// TIA Portal V20 export
DATA_BLOCK "EmNodes"   // DB146
// Global DB for the data exchange between the module levels (Between Unit and EM or EM and CM)
// stored: Access Published, MemoryReserve 100, Namespace Unit1
   VAR
      unitStatus { ExternalWritable := 'False'} : "LAF_typeUnitStatus";   // Status of the unit
      emFeedback { ExternalWritable := 'False'} : Array[0.._.U1_NO_OF_EMs] of "LUC_typeEmFeedback";   // Status of the individual equipment modules
      emRelations { ExternalWritable := 'False'} : "Unit1.LER_typeEmRelation";
      emIt { S7_SetPoint := 'True'} : Array[0..13] of "LER_OEM_Data";
      enableControlInterfaces { ExternalWritable := 'False'} : "LAF_typeEnableControlInterfaces";
      oem { ExternalAccessible := 'False'; ExternalVisible := 'False'; ExternalWritable := 'False'; S7_SetPoint := 'True'} : Array[0..10] of "LER_OEM_Data";
      FATModeSelect { ExternalWritable := 'False'} : "LER_TypeFATMode_ModeSelect";
   END_VAR
   VAR RETAIN
      FATModeInterface { ExternalWritable := 'False'} : "LER_TypeFATModeInterface";
   END_VAR
   VAR
      signalStack { ExternalWritable := 'False'} : "LUC_typeSignalStackByBool";
      clock { ExternalWritable := 'False'} : "LAF_typeGlobalClockMem";
      slmRunning { ExternalWritable := 'False'} : Bool;
      slmPowerOff { ExternalWritable := 'False'} : Bool;
      InterfaceTestMode { ExternalWritable := 'False'} : Bool;
      CapabilityModeComplete { ExternalWritable := 'False'} : Bool;
      SamplingModeComplete { ExternalWritable := 'False'} : Bool;
      stateCommandsExecute { ExternalWritable := 'False'} : Bool;
      atLeastOneDoorUnLock { ExternalWritable := 'False'} : Bool;
      SleepModeActivationTime { ExternalWritable := 'False'} : Time;
      DeepSleepModeActivationTime { ExternalWritable := 'False'} : Time;
      SleepModeChangeReq { ExternalWritable := 'False'} : Bool;
      DeepSleepModeChangeReq { ExternalWritable := 'False'} : Bool;
      WakeupRecoveryRequired { ExternalWritable := 'False'} : Bool;
      "========Communication========" { ExternalWritable := 'False'} : Bool;
      BA030 { ExternalWritable := 'False'} : "LER_typeCommunication";
      BA040 { ExternalWritable := 'False'} : "LER_typeCommunication";
      "========Safety========" { ExternalWritable := 'False'} : Bool;
      devicesSummary { ExternalWritable := 'False'} : "LWONIK_typeDevicesStatusSummary";
      OperationMode { ExternalWritable := 'False'} : "LWONIK_typeOperationMode";
      PhmiMode { ExternalWritable := 'False'} : "LWONIK_typePhmiMode";
      ScsMode { ExternalWritable := 'False'} : "LWONIK_typeScsMode";
      RcMode1 { ExternalWritable := 'False'} : "LWONIK_typeRollChangeMode";
      RcMode2 { ExternalWritable := 'False'} : "LWONIK_typeRollChangeMode";
      SafetyZone1OpEnable { ExternalWritable := 'False'} : "LWONIK_typeSafetyZoneManualOperation";
      SafetyZone2OpEnable { ExternalWritable := 'False'} : "LWONIK_typeSafetyZoneManualOperation";
      SafetyZone3OpEnable { ExternalWritable := 'False'} : "LWONIK_typeSafetyZoneManualOperation";
      Zone1SafetyStatus { ExternalWritable := 'False'} : "LWONIK_typeZoneStatus";
      Zone2SafetyStatus { ExternalWritable := 'False'} : "LWONIK_typeZoneStatus";
      Zone3SafetyStatus { ExternalWritable := 'False'} : "LWONIK_typeZoneStatus";
      SafetySensor { ExternalWritable := 'False'} : "LWONIK_typeSafetySensor";
      EstopStatus { ExternalWritable := 'False'} : "LWONIK_typeFromSafetyEstopStatus";
      FdoorStatus { ExternalWritable := 'False'} : "LWONIK_typeFromSafetyDoorStatus";
      MobilePanelConnected { ExternalWritable := 'False'} : Bool;
      EnableACK { ExternalWritable := 'False'} : Bool;
      SS1Extention { ExternalWritable := 'False'} : Bool;
      LHSS1Extention { ExternalWritable := 'False'} : Bool;
      RHSS1Extention { ExternalWritable := 'False'} : Bool;
      LH_RollChangeActive { ExternalWritable := 'False'} : Bool;
      RH_RollChangeActive { ExternalWritable := 'False'} : Bool;
      Z_FOLD_AllEstopsOK { ExternalWritable := 'False'} : Bool;
      "=======ETC========" { ExternalWritable := 'False'} : Bool;
   END_VAR
   VAR RETAIN
      unitRecipe { ExternalWritable := 'False'} : "Unit1.typeRecipe";
   END_VAR
   VAR
      unitCycleTime { ExternalWritable := 'False'} : Time;
      "unitCycleTime/2" { ExternalWritable := 'False'} : Time;
      "unitCycleTime/6" { ExternalWritable := 'False'} : Time;
      allBrakeTest { ExternalWritable := 'False'} : "LER_typeBrakeTestUnitInterface";
      HourTestModeAllOK { ExternalWritable := 'False'} : Bool;
      CapabilityModeAllOK { ExternalWritable := 'False'} : Bool;
      ScrapBox { ExternalWritable := 'False'} : Struct
         LockSW : Bool;
         UnlockSW : Bool;
         ResetSW : Bool;
      END_STRUCT;
      LeftSafeScale { ExternalWritable := 'False'} : Int := 120;
      RightSafeScale { ExternalWritable := 'False'} : Int := 120;
      LeftMaxValue : Int := 1020;
      RightMaxValue : Int := 1020;
   END_VAR
BEGIN
   // BA030.ReelCutToStack.InterfaceData."Bool"[0] : To Load Enable
   // BA030.ReelCutToStack.InterfaceData."Bool"[1] : To Load Complete Comfirm
   // BA030.ReelCutToStack.InterfaceData."Bool"[2] : Cell Data Report
   // BA030.ReelCutToStack.InterfaceData."Bool"[10] : CollisionAreaOn
   // BA030.ReelCutToStack.InterfaceData."Bool"[11] : CollisionAreaOff
   // BA030.ReelCutToStack.InterfaceData."Bool"[15] : HeartBeat
   // BA030.ReelCutToStack.InterfaceData."Bool"[20] : To ReelCut Motion Ready Status (ReelCut Full)
   // BA030.ReelCutToStack.InterfaceData."Bool"[21] : To ReelCut in Motion Auto Standby
   // BA030.ReelCutToStack.InterfaceData."Bool"[22] : To ReelCut in Motion Auto Mode
   // BA030.ReelCutToStack.InterfaceData."Bool"[23] : To Motion Stop CMD (Motion Stop Req)
   // BA030.ReelCutToStack.InterfaceData."Bool"[30] : HoursTestMode.On/Off.Status (ReelCut)
   // BA030.ReelCutToStack.InterfaceData."Bool"[31] : HourTestMode_Completed (ReelCut)
   // BA030.ReelCutToStack.InterfaceData."Bool"[32] : CapabilityMode.On/Off.Status (ReelCut)
   // BA030.ReelCutToStack.InterfaceData."Bool"[33] : CapabilityMode_Completed (ReelCut)
   // BA030.ReelCutToStack.InterfaceData."Bool"[34] : FATMode.Apply (ReelCut)
   // BA030.ReelCutToStack.InterfaceData.LReal[10] : Select Hours (ReelCut)
   // BA030.StackToReelCut.UnitStatus.specialFunctions.SingleMode : Not Use Stack1
   // BA030.StackToReelCut.InterfaceData."Bool"[0] : From Load Requset
   // BA030.StackToReelCut.InterfaceData."Bool"[1] : From Load Busy
   // BA030.StackToReelCut.InterfaceData."Bool"[2] : From Load Complete
   // BA030.StackToReelCut.InterfaceData."Bool"[3] : Cell Data Request
   // BA030.StackToReelCut.InterfaceData."Bool"[4] : Cell Data Report Ack
   // BA030.StackToReelCut.InterfaceData."Bool"[5] : Cell Data Report Nck
   // BA030.StackToReelCut.InterfaceData."Bool"[10] : Stack#1 Gauge RnR Complete
   // BA030.StackToReelCut.InterfaceData."Bool"[15] : HeartBeat
   // BA030.StackToReelCut.InterfaceData."Bool"[19] : From Stack#1 Count Mismatch Call
   // BA030.StackToReelCut.InterfaceData."Bool"[20] : From Motion Ready Status (Stack#1 Full)
   // BA030.StackToReelCut.InterfaceData."Bool"[21] : From Stack#1 in Motion Auto Standby
   // BA030.StackToReelCut.InterfaceData."Bool"[22] : From Stack#1 in Motion Auto Mode
   // BA030.StackToReelCut.InterfaceData."Bool"[23] : From Motion Start CMD (Stack#1 Motion Req)
   // BA030.StackToReelCut.InterfaceData."Bool"[24] : From Motion Stop CMD (Stack#1 Error)
   // BA030.StackToReelCut.InterfaceData."Bool"[25] : From Stack#1 Unloading
   // BA030.StackToReelCut.InterfaceData."Bool"[26] : From Stack#1 Loading Ok
   // BA030.StackToReelCut.InterfaceData."Bool"[30] : HoursTestMode.On/Off.Status (STK1)
   // BA030.StackToReelCut.InterfaceData."Bool"[31] : HourTestMode_Completed (STK1)
   // BA030.StackToReelCut.InterfaceData."Bool"[32] : CapabilityMode.On/Off.Status (STK1)
   // BA030.StackToReelCut.InterfaceData."Bool"[33] : CapabilityMode_Completed (STK1)
   // BA030.StackToReelCut.InterfaceData."Bool"[34] : FATMode.Apply (STK1)
   // BA030.StackToReelCut.InterfaceData."Bool"[40] : HoursTestMode.On/Off.Status (INS)
   // BA030.StackToReelCut.InterfaceData."Bool"[41] : HourTestMode_Completed (INS)
   // BA030.StackToReelCut.InterfaceData."Bool"[42] : CapabilityMode.On/Off.Status (INS)
   // BA030.StackToReelCut.InterfaceData."Bool"[43] : CapabilityMode_Completed (INS)
   // BA030.StackToReelCut.InterfaceData."Bool"[44] : FATMode.Apply (INS)
   // BA030.StackToReelCut.InterfaceData."Bool"[50] : HoursTestMode.On/Off.Status (ReelCut10)
   // BA030.StackToReelCut.InterfaceData."Bool"[51] : HourTestMode_Completed (ReelCut10)
   // BA030.StackToReelCut.InterfaceData."Bool"[52] : CapabilityMode.On/Off.Status (ReelCut10)
   // BA030.StackToReelCut.InterfaceData."Bool"[53] : CapabilityMode_Completed (ReelCut10)
   // BA030.StackToReelCut.InterfaceData."Bool"[54] : FATMode.Apply (ReelCut10)
   // BA030.StackToReelCut.InterfaceData."Bool"[60] : HoursTestMode.On/Off.Status (ReelCut15)
   // BA030.StackToReelCut.InterfaceData."Bool"[61] : HourTestMode_Completed (ReelCut15)
   // BA030.StackToReelCut.InterfaceData."Bool"[62] : CapabilityMode.On/Off.Status (ReelCut15)
   // BA030.StackToReelCut.InterfaceData."Bool"[63] : CapabilityMode_Completed (ReelCut15)
   // BA030.StackToReelCut.InterfaceData."Bool"[64] : FATMode.Apply (ReelCut15)
   // BA030.StackToReelCut.InterfaceData.LReal[0] : From Stack#1 Cell Count
   // BA030.StackToReelCut.InterfaceData.LReal[1] : From Stack#1 CPM
   // BA030.StackToReelCut.InterfaceData.LReal[2] : Stack#1 Gauge RnR3 Mode Count
   // BA030.StackToReelCut.InterfaceData.LReal[10] : Select Hours (STK)
   // BA030.StackToReelCut.InterfaceData.LReal[11] : Select Hours (INS)
   // BA030.StackToReelCut.InterfaceData.LReal[12] : Select Hours (ReelCut10)
   // BA030.StackToReelCut.InterfaceData.LReal[13] : Select Hours (ReelCut15)
   // BA030.StackToReelCut.InterfaceData.LReal[14] : Capability Count Current
   // BA030.StackToReelCut.InterfaceData.LReal[15] : Capability Count Set
   // BA040.ReelCutToStack.InterfaceData."Bool"[0] : To Load Enable
   // BA040.ReelCutToStack.InterfaceData."Bool"[1] : To Load Complete Comfirm
   // BA040.ReelCutToStack.InterfaceData."Bool"[2] : Cell Data Report
   // BA040.ReelCutToStack.InterfaceData."Bool"[10] : CollisionAreaOn
   // BA040.ReelCutToStack.InterfaceData."Bool"[11] : CollisionAreaOff
   // BA040.ReelCutToStack.InterfaceData."Bool"[15] : HeartBeat
   // BA040.ReelCutToStack.InterfaceData."Bool"[20] : To ReelCut Motion Ready Status(ReelCut Full)
   // BA040.ReelCutToStack.InterfaceData."Bool"[21] : To ReelCut in Motion Auto Standby
   // BA040.ReelCutToStack.InterfaceData."Bool"[22] : To ReelCut in Motion Auto Mode
   // BA040.ReelCutToStack.InterfaceData."Bool"[23] : To Motion Stop CMD (Motion Stop Req)
   // BA040.ReelCutToStack.InterfaceData."Bool"[30] : HoursTestMode.On/Off.Status (ReelCut)
   // BA040.ReelCutToStack.InterfaceData."Bool"[31] : HourTestMode_Completed (ReelCut)
   // BA040.ReelCutToStack.InterfaceData."Bool"[32] : CapabilityMode.On/Off.Status (ReelCut)
   // BA040.ReelCutToStack.InterfaceData."Bool"[33] : CapabilityMode_Completed (ReelCut)
   // BA040.ReelCutToStack.InterfaceData."Bool"[34] : FATMode.Apply (ReelCut)
   // BA040.ReelCutToStack.InterfaceData.LReal[10] : Select Hours (ReelCut)
   // BA040.StackToReelCut.UnitStatus.specialFunctions.SingleMode : Not Use Stack2
   // BA040.StackToReelCut.InterfaceData."Bool"[0] : From Load Requset
   // BA040.StackToReelCut.InterfaceData."Bool"[1] : From Load Busy
   // BA040.StackToReelCut.InterfaceData."Bool"[2] : From Load Complete
   // BA040.StackToReelCut.InterfaceData."Bool"[3] : Cell Data Request
   // BA040.StackToReelCut.InterfaceData."Bool"[4] : Cell Data Report Ack
   // BA040.StackToReelCut.InterfaceData."Bool"[5] : Cell Data Report Nck
   // BA040.StackToReelCut.InterfaceData."Bool"[10] : Stack#2 Gauge RnR Complete
   // BA040.StackToReelCut.InterfaceData."Bool"[15] : HeartBeat
   // BA040.StackToReelCut.InterfaceData."Bool"[19] : From Stack#2 Count Mismatch Call
   // BA040.StackToReelCut.InterfaceData."Bool"[20] : From Motion Ready Status (Stack#2 Full)
   // BA040.StackToReelCut.InterfaceData."Bool"[21] : From Stack#2 in Motion Auto Standby
   // BA040.StackToReelCut.InterfaceData."Bool"[22] : From Stack#2 in Motion Auto Mode
   // BA040.StackToReelCut.InterfaceData."Bool"[23] : From Motion Start CMD (Stack#2 Motion Req)
   // BA040.StackToReelCut.InterfaceData."Bool"[24] : From Motion Stop CMD (Stack#2 Error)
   // BA040.StackToReelCut.InterfaceData."Bool"[25] : From Stack#2 Unloading
   // BA040.StackToReelCut.InterfaceData."Bool"[26] : From Stack#2 Loading Ok
   // BA040.StackToReelCut.InterfaceData."Bool"[30] : HoursTestMode.On/Off.Status (STK2)
   // BA040.StackToReelCut.InterfaceData."Bool"[31] : HourTestMode_Completed (STK2)
   // BA040.StackToReelCut.InterfaceData."Bool"[32] : CapabilityMode.On/Off.Status (STK2)
   // BA040.StackToReelCut.InterfaceData."Bool"[33] : CapabilityMode_Completed (STK2)
   // BA040.StackToReelCut.InterfaceData."Bool"[34] : FATMode.Apply (STK2)
   // BA040.StackToReelCut.InterfaceData."Bool"[40] : HoursTestMode.On/Off.Status (INS)
   // BA040.StackToReelCut.InterfaceData."Bool"[41] : HourTestMode_Completed (INS)
   // BA040.StackToReelCut.InterfaceData."Bool"[42] : CapabilityMode.On/Off.Status (INS)
   // BA040.StackToReelCut.InterfaceData."Bool"[43] : CapabilityMode_Completed (INS)
   // BA040.StackToReelCut.InterfaceData."Bool"[44] : FATMode.Apply (INS)
   // BA040.StackToReelCut.InterfaceData."Bool"[50] : HoursTestMode.On/Off.Status (ReelCut10)
   // BA040.StackToReelCut.InterfaceData."Bool"[51] : HourTestMode_Completed (ReelCut10)
   // BA040.StackToReelCut.InterfaceData."Bool"[52] : CapabilityMode.On/Off.Status (ReelCut10)
   // BA040.StackToReelCut.InterfaceData."Bool"[53] : CapabilityMode_Completed (ReelCut10)
   // BA040.StackToReelCut.InterfaceData."Bool"[54] : FATMode.Apply (ReelCut10)
   // BA040.StackToReelCut.InterfaceData."Bool"[60] : HoursTestMode.On/Off.Status (ReelCut15)
   // BA040.StackToReelCut.InterfaceData."Bool"[61] : HourTestMode_Completed (ReelCut15)
   // BA040.StackToReelCut.InterfaceData."Bool"[62] : CapabilityMode.On/Off.Status (ReelCut15)
   // BA040.StackToReelCut.InterfaceData."Bool"[63] : CapabilityMode_Completed (ReelCut15)
   // BA040.StackToReelCut.InterfaceData."Bool"[64] : FATMode.Apply (ReelCut15)
   // BA040.StackToReelCut.InterfaceData.LReal[0] : From Stack#2 Cell Count
   // BA040.StackToReelCut.InterfaceData.LReal[1] : From Stack#2 CPM
   // BA040.StackToReelCut.InterfaceData.LReal[2] : Stack#2 Gauge RnR3 Mode Count
   // BA040.StackToReelCut.InterfaceData.LReal[10] : Select Hours (STK)
   // BA040.StackToReelCut.InterfaceData.LReal[11] : Select Hours (INS)
   // BA040.StackToReelCut.InterfaceData.LReal[12] : Select Hours (ReelCut10)
   // BA040.StackToReelCut.InterfaceData.LReal[13] : Select Hours (ReelCut15)
   // BA040.StackToReelCut.InterfaceData.LReal[14] : Capability Count Current
   // BA040.StackToReelCut.InterfaceData.LReal[15] : Capability Count Set
   unitRecipe.processUnitNo := 2;
   // allBrakeTest.monitoring.emStatus.axisEnabled[0] : cmUnwinderAxisEm0
   // allBrakeTest.monitoring.emStatus.axisEnabled[1] : cmUnwinderAxisEm1
   // allBrakeTest.monitoring.emStatus.axisEnabled[2] : cmCompensatorAxis
   // allBrakeTest.monitoring.emStatus.axisEnabled[3] : cmFeedingRollAxis
   // allBrakeTest.monitoring.emStatus.axisEnabled[4] : cmCutterAxis
   // allBrakeTest.monitoring.emStatus.axisEnabled[5] : cmPositionMovingAxis
   // allBrakeTest.monitoring.emStatus.axisEnabled[6] : cmMagazineAxis
   // allBrakeTest.monitoring.emStatus.axisEnabled[7] : cmVisionAxis
   // allBrakeTest.monitoring.emStatus.axisEnabled[8] : cmNgKickerAxis
   // allBrakeTest.monitoring.emStatus.axisEnabled[9] : cmPassKickerAxis
   // allBrakeTest.monitoring.emStatus.busy[0] : cmUnwinderAxisEm0
   // allBrakeTest.monitoring.emStatus.busy[1] : cmUnwinderAxisEm1
   // allBrakeTest.monitoring.emStatus.busy[2] : cmCompensatorAxis
   // allBrakeTest.monitoring.emStatus.busy[3] : cmFeedingRollAxis
   // allBrakeTest.monitoring.emStatus.busy[4] : cmCutterAxis
   // allBrakeTest.monitoring.emStatus.busy[5] : cmPositionMovingAxis
   // allBrakeTest.monitoring.emStatus.busy[6] : cmMagazineAxis
   // allBrakeTest.monitoring.emStatus.busy[7] : cmVisionAxis
   // allBrakeTest.monitoring.emStatus.busy[8] : cmNgKickerAxis
   // allBrakeTest.monitoring.emStatus.busy[9] : cmPassKickerAxis
   // allBrakeTest.monitoring.emStatus.complete[0] : cmUnwinderAxisEm0
   // allBrakeTest.monitoring.emStatus.complete[1] : cmUnwinderAxisEm1
   // allBrakeTest.monitoring.emStatus.complete[2] : cmCompensatorAxis
   // allBrakeTest.monitoring.emStatus.complete[3] : cmFeedingRollAxis
   // allBrakeTest.monitoring.emStatus.complete[4] : cmCutterAxis
   // allBrakeTest.monitoring.emStatus.complete[5] : cmPositionMovingAxis
   // allBrakeTest.monitoring.emStatus.complete[6] : cmMagazineAxis
   // allBrakeTest.monitoring.emStatus.complete[7] : cmVisionAxis
   // allBrakeTest.monitoring.emStatus.complete[8] : cmNgKickerAxis
   // allBrakeTest.monitoring.emStatus.complete[9] : cmPassKickerAxis
   // allBrakeTest.monitoring.error : Brake Test Error
   // allBrakeTest.monitoring.allBusy : Brake Test In Progress
   // allBrakeTest.monitoring.allComplete : Brake Test Done
END_DATA_BLOCK
